FUNCTION_BLOCK XTSIOEnvVarWrapper
VAR
	XtsIoEnvironment : Tc3_XTS_Utility.FB_TcIoXtsEnvironment;
	XPU: Tc3_XTS_Utility.I_TcIoXtsProcessingUnit;
END_VAR

METHOD GetCaGroupInterface : I_Mc2CaGroup
VAR_INPUT
	CAGroupNumber : INT;
END_VAR
GetCaGroupInterface := XtsIoEnvironment.Mc2CaGroup(CAGroupNumber);
END_METHOD

METHOD PUBLIC GetMotorModuleInterface : I_TcIoXtsPartModule
VAR_INPUT
	PartNumber : INT;
	ModuleNumber : INT;
END_VAR
XPU.PartTcIo(PartNumber).ModuleTcIo(ModuleNumber);
END_METHOD

METHOD PUBLIC GetMoverInterface : I_TcIoXtsXpuMover
VAR_INPUT
	MoverId : INT;
END_VAR
GetMoverInterface := XPU.MoverTcIo(MoverID);
END_METHOD

METHOD PUBLIC GetPartInterface : I_TcIoXtsXpuPart
VAR_INPUT
	PartNumber : INT;
END_VAR
GetPartInterface := XPU.PartTcIo(PartNumber);
END_METHOD

METHOD PUBLIC GetTrackInterface : I_TcIoXtsXpuTrack
VAR_INPUT
	TrackNumber : INT;
END_VAR
GetTrackInterface := XPU.TrackTcIo(TrackNumber);
END_METHOD

METHOD PUBLIC Initialise : BOOL
VAR_INPUT
END_VAR
IF XtsIoEnvironment.Init(TRUE) THEN
	XtsIoEnvironment.Init(FALSE);
	XPU := XtsIoEnvironment.XpuTcIo(1);
	Initialise := TRUE;
END_IF
END_METHOD

END_FUNCTION_BLOCK

(* stored: Version 1.1.0.1, ProductVersion 3.1.4024.12
   POU XTSIOEnvVarWrapper: Id {03c3c931-6ee3-4ab9-88b9-320f3e1d8e15}, SpecialFunc None
   Method GetCaGroupInterface: Id {12f834a0-9ae6-48b5-9bae-7bc717cd2b2d}
   Method GetMotorModuleInterface: Id {9af7c768-b524-4dfc-b4c9-d134e43969ae}
   Method GetMoverInterface: Id {dbc9b774-d169-476b-835b-9bf55e4a60d9}
   Method GetPartInterface: Id {a60c8186-f31f-4591-b959-ebb1bad32c7a}
   Method GetTrackInterface: Id {36334a76-598d-4a99-aaef-0a407eed48bd}
   Method Initialise: Id {f0d17991-21f7-403c-899a-0fcccbff041e} *)
